FUNCTION_BLOCK Server
  (* Standard: 61499-2 *)
  (* Version 0.2, 2003-12-04, JHC, Rockwell Automation, Renamed for better indexing. *)
  (* Version 0.1, 2002-11-05, JHC, Rockwell Automation, Corrected missing ST element in Algorithm REQ. *)
  (* Version 0.0, 2000-05-30, JHC, Rockwell Automation *)
  (* Compiler header: package fb.rt.cs725; *)
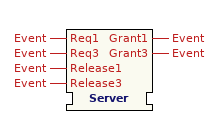
  EVENT_INPUT
    Req1;
    Req3; (* Normal Execution Request *)
    Release1;
    Release3;
  END_EVENT
  EVENT_OUTPUT
    Grant1;
    Grant3;
  END_EVENT
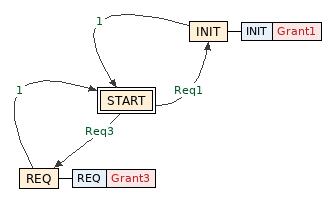
  EC_STATES
    START; (* Initial State *)
    INIT : INIT -> Grant1; (* Initialization *)
    REQ : REQ -> Grant3; (* Normal execution *)
  END_STATES
  EC_TRANSITIONS
    START TO INIT := Req1;
    INIT TO START := 1;
    START TO REQ := Req3;
    REQ TO START := 1;
  END_TRANSITIONS
  ALGORITHM INIT IN ST: (* Initialization algorithm *)

  END_ALGORITHM
  ALGORITHM REQ IN ST: (* Normally executed algorithm *)

  END_ALGORITHM
END_FUNCTION_BLOCK
